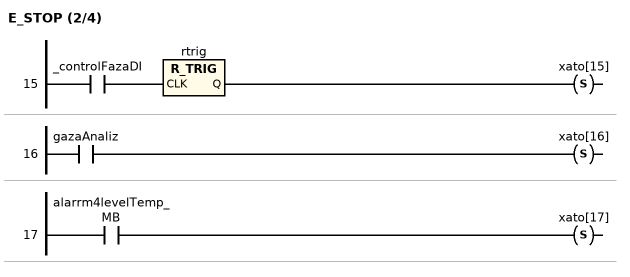
[picture p24: E_STOP (LD)]
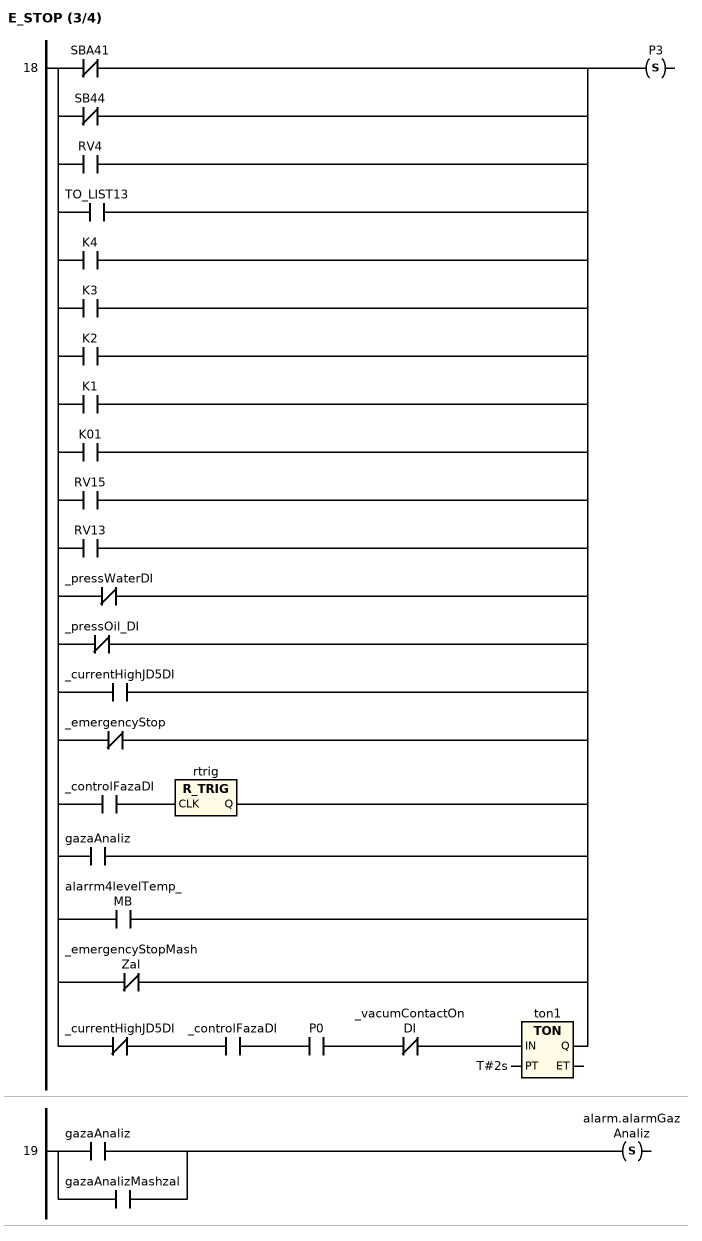
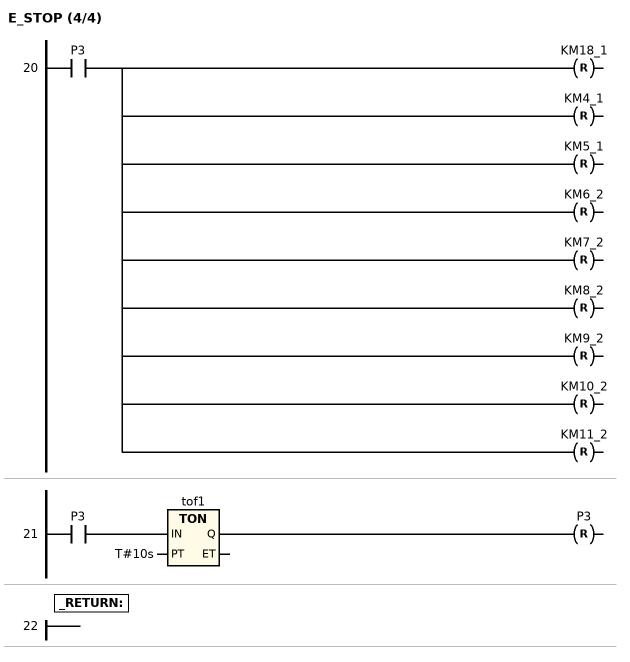
_LD_ (* Ladder Diagram *)
NETWORK 1
	[/SBA41] --- (S xato[0])
NETWORK 2
	[rv4] --- (S xato[1])
NETWORK 3
	[TO_LIST13] --- (S xato[2])
NETWORK 4
	[k4] --- (S xato[3])
NETWORK 5
	[k3] --- (S xato[4])
NETWORK 6
	[k2] --- (S xato[5])
NETWORK 7
	[k1] --- (S xato[6])
NETWORK 8
	[k01] --- (S xato[7])
NETWORK 9
	[rv15] --- (S xato[8])
NETWORK 10
	[rv13] --- (S xato[9])
NETWORK 11
	[/_pressWaterDI] --- (S xato[10])
NETWORK 12
	[/_pressOil_DI] --- (S xato[11])
NETWORK 13
	[/_currentHighJD5DI] --- (S xato[13])
NETWORK 14
	[/_emergencyStop] --- (S xato[14])
NETWORK 15
	[_controlFazaDI] - rtrig:R_TRIG(CLK: *) --- (S xato[15])
NETWORK 16
	[gazaAnaliz] --- (S xato[16])
NETWORK 17
	[alarrm4levelTemp_MB] --- (S xato[17])
NETWORK 18
	{ [/SBA41] | [/SB44] | [RV4] | [TO_LIST13] | [K4] | [K3] | [K2] | [K1] | [K01] | [RV15] | [RV13] | [/_pressWaterDI] | [/_pressOil_DI] | [_currentHighJD5DI] | [/_emergencyStop] | [_controlFazaDI] - rtrig:R_TRIG(CLK: *) | [gazaAnaliz] | [alarrm4levelTemp_MB] | [/_emergencyStopMashZal] | [/_currentHighJD5DI] - [_controlFazaDI] - [P0] - [/_vacumContactOnDI] - ton1:TON(IN: *, PT: T#2s) } --- (S P3)
NETWORK 19
	{ [gazaAnaliz] | [gazaAnalizMashzal] } --- (S alarm.alarmGazAnaliz)
NETWORK 20
	[P3] --- (R KM18_1) (R KM4_1) (R KM5_1) (R KM6_2) (R KM7_2) (R KM8_2) (R KM9_2) (R KM10_2) (R KM11_2)
NETWORK 21
	[P3] - tof1:TON(IN: *, PT: T#10s) --- (R P3)
NETWORK 22 _RETURN::
	*
_END_LD_
(* the same logic as Structured Text *)
(* Network 1 *)
IF NOT SBA41 THEN xato[0] := TRUE; END_IF;
(* Network 2 *)
IF rv4 THEN xato[1] := TRUE; END_IF;
(* Network 3 *)
IF TO_LIST13 THEN xato[2] := TRUE; END_IF;
(* Network 4 *)
IF k4 THEN xato[3] := TRUE; END_IF;
(* Network 5 *)
IF k3 THEN xato[4] := TRUE; END_IF;
(* Network 6 *)
IF k2 THEN xato[5] := TRUE; END_IF;
(* Network 7 *)
IF k1 THEN xato[6] := TRUE; END_IF;
(* Network 8 *)
IF k01 THEN xato[7] := TRUE; END_IF;
(* Network 9 *)
IF rv15 THEN xato[8] := TRUE; END_IF;
(* Network 10 *)
IF rv13 THEN xato[9] := TRUE; END_IF;
(* Network 11 *)
IF NOT _pressWaterDI THEN xato[10] := TRUE; END_IF;
(* Network 12 *)
IF NOT _pressOil_DI THEN xato[11] := TRUE; END_IF;
(* Network 13 *)
IF NOT _currentHighJD5DI THEN xato[13] := TRUE; END_IF;
(* Network 14 *)
IF NOT _emergencyStop THEN xato[14] := TRUE; END_IF;
(* Network 15 *)
rtrig(CLK := _controlFazaDI);
IF rtrig.Q THEN xato[15] := TRUE; END_IF;
(* Network 16 *)
IF gazaAnaliz THEN xato[16] := TRUE; END_IF;
(* Network 17 *)
IF alarrm4levelTemp_MB THEN xato[17] := TRUE; END_IF;
(* Network 18 *)
rtrig(CLK := _controlFazaDI);
ton1(IN := NOT _currentHighJD5DI AND _controlFazaDI AND P0 AND NOT _vacumContactOnDI, PT := T#2s);
IF NOT SBA41 OR NOT SB44 OR RV4 OR TO_LIST13 OR K4 OR K3 OR K2 OR K1 OR K01 OR RV15 OR RV13 OR NOT _pressWaterDI OR NOT _pressOil_DI OR _currentHighJD5DI OR NOT _emergencyStop OR rtrig.Q OR gazaAnaliz OR alarrm4levelTemp_MB OR NOT _emergencyStopMashZal OR ton1.Q THEN P3 := TRUE; END_IF;
(* Network 19 *)
IF gazaAnaliz OR gazaAnalizMashzal THEN alarm.alarmGazAnaliz := TRUE; END_IF;
(* Network 20 *)
IF P3 THEN KM18_1 := FALSE; KM4_1 := FALSE; KM5_1 := FALSE; KM6_2 := FALSE; KM7_2 := FALSE; KM8_2 := FALSE; KM9_2 := FALSE; KM10_2 := FALSE; KM11_2 := FALSE; END_IF;
(* Network 21 *)
tof1(IN := P3, PT := T#10s);
IF tof1.Q THEN P3 := FALSE; END_IF;
(* Network 22 *)
(* label: _RETURN: *)
END_PROGRAM

(* POU blink, CFC *)
PROGRAM blink
VAR
	tp1: TP;
	tp2: TP;
	out: BOOL;
	vaqt : TIME := T#500ms;
END_VAR
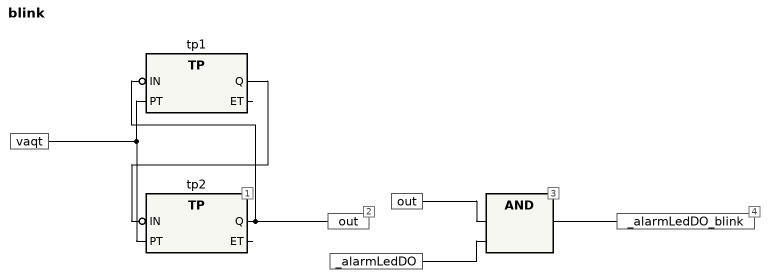
_CFC_ (* Continuous Function Chart, elements in execution order *)
#0 tp1:TP(IN: NOT #1.Q, PT: vaqt)
#1 tp2:TP(IN: NOT #0.Q, PT: vaqt)
#2 out <= #1.Q
#3 AND(out, _alarmLedDO)
#4 _alarmLedDO_blink <= #3
_END_CFC_
(* the same logic as Structured Text *)
tp1(IN := NOT tp2.Q, PT := vaqt);
tp2(IN := NOT tp1.Q, PT := vaqt);
out := tp2.Q;
_alarmLedDO_blink := out AND _alarmLedDO;
END_PROGRAM

(* Visualisation main
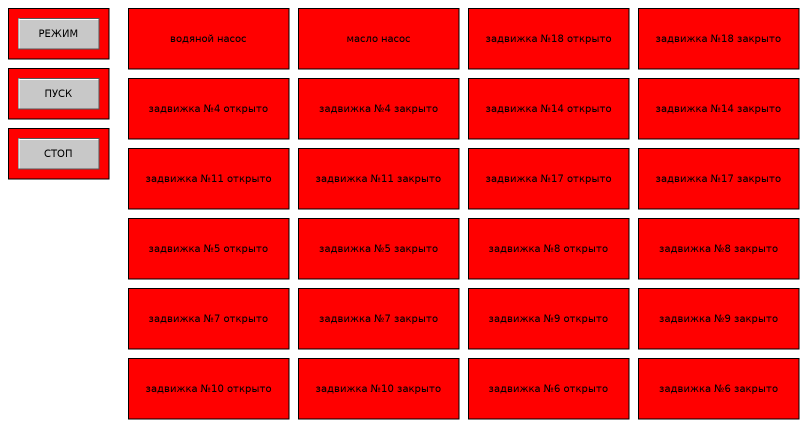
rounded rectangle at (130,10)-(291,71): text "водяной насос"; alarm colour if .KM1
rounded rectangle at (300,10)-(461,71): text "масло насос"; alarm colour if .KM2
rounded rectangle at (470,10)-(631,71): text "задвижка №18 открыто"; alarm colour if .KM18_1
rounded rectangle at (640,10)-(801,71): text "задвижка №18 закрыто"; alarm colour if .KM18_2
rounded rectangle at (130,80)-(291,141): text "задвижка №4 открыто"; alarm colour if .KM4_1
rounded rectangle at (300,80)-(461,141): text "задвижка №4 закрыто"; alarm colour if ._4gate.closed
rounded rectangle at (470,80)-(631,141): text "задвижка №14 открыто"; alarm colour if ._14gate.opened
rounded rectangle at (640,80)-(801,141): text "задвижка №14 закрыто"; alarm colour if ._14gate.closed
rounded rectangle at (130,150)-(291,211): text "задвижка №11 открыто"; alarm colour if ._11gate.opened
rounded rectangle at (300,150)-(461,211): text "задвижка №11 закрыто"; alarm colour if ._11gate.closed
rounded rectangle at (470,150)-(631,211): text "задвижка №17 открыто"; alarm colour if ._17gate.opened
rounded rectangle at (640,150)-(801,211): text "задвижка №17 закрыто"; alarm colour if ._17gate.closed
rounded rectangle at (130,220)-(291,281): text "задвижка №5 открыто"; alarm colour if ._5gate.opened
rounded rectangle at (300,220)-(461,281): text "задвижка №5 закрыто"; alarm colour if ._5gate.closed
rounded rectangle at (470,220)-(631,281): text "задвижка №8 открыто"; alarm colour if ._8gate.opened
rounded rectangle at (640,220)-(801,281): text "задвижка №8 закрыто"; alarm colour if ._8gate.closed
rounded rectangle at (130,290)-(291,351): text "задвижка №7 открыто"; alarm colour if ._7gate.opened
rounded rectangle at (300,290)-(461,351): text "задвижка №7 закрыто"; alarm colour if ._7gate.closed
rounded rectangle at (470,290)-(631,351): text "задвижка №9 открыто"; alarm colour if ._9gate.opened
rounded rectangle at (640,290)-(801,351): text "задвижка №9 закрыто"; alarm colour if ._9gate.closed
rounded rectangle at (130,360)-(291,421): text "задвижка №10 открыто"; alarm colour if ._10gate.opened
rounded rectangle at (300,360)-(461,421): text "задвижка №10 закрыто"; alarm colour if ._10gate.closed
rounded rectangle at (470,360)-(631,421): text "задвижка №6 открыто"; alarm colour if ._6gate.opened
rounded rectangle at (640,360)-(801,421): text "задвижка №6 закрыто"; alarm colour if ._6gate.closed
rounded rectangle at (10,130)-(111,181): alarm colour if .goSTOP
button at (20,140)-(101,171): text "СТОП"; toggles .SB53_1
rounded rectangle at (10,70)-(111,121): alarm colour if .goPusk
button at (20,80)-(101,111): text "ПУСК"; toggles .SB43
rounded rectangle at (10,10)-(111,61): alarm colour if .goRejim
button at (20,20)-(101,51): text "РЕЖИМ"; toggles .SB42
*)
